# EPICS substitutions: lensApp/Db/stacklens1.substitutions
file stacklens1.tpl-db
{
    {
        LOCATION = $(LOCATION)
        MOTID    = $(MOTID)
        LENSID   = $(LENSID)
    }
}

file stacklens.tpl-db
{
    {
        LOCATION = $(LOCATION)
        MOTID    = $(MOTID)
        Y_MOT    = $(Y_MOT)
    }
}

file lensMotion.tpl-db
{
    {
        LOCATION = $(LOCATION)
        MOTID    = $(MOTID)
        Y_MOT    = $(Y_MOT)
        LENSID   = $(LENSID)
        IN_STATE = $(IN_STATE)
    }
}
